FUNCTION COSD : LREAL
VAR_INPUT
	ANGLE:LREAL;
END_VAR
VAR
END_VAR

COSD:=COS(DEG_TO_RAD(ANGLE));

END_FUNCTION

(* stored: Version 1.1.0.1, ProductVersion 3.1.4024.12
   POU COSD: Id {bb736399-f365-4fea-b648-f1576e601419}, SpecialFunc None *)
